(* PLC project PLC_1, BaoSight BAOSKY 2.0 *)
(* stored: creationDateTime 2026-09-22T15:06:44.776 *)

PROGRAM PU_1
  VAR
    aa : DWORD := 0001;
  END_VAR

 aa := ROR(IN:=aa,N:=1);
END_PROGRAM

CONFIGURATION PLC_Task
  RESOURCE PLC_Task ON PLC
  END_RESOURCE
END_CONFIGURATION
